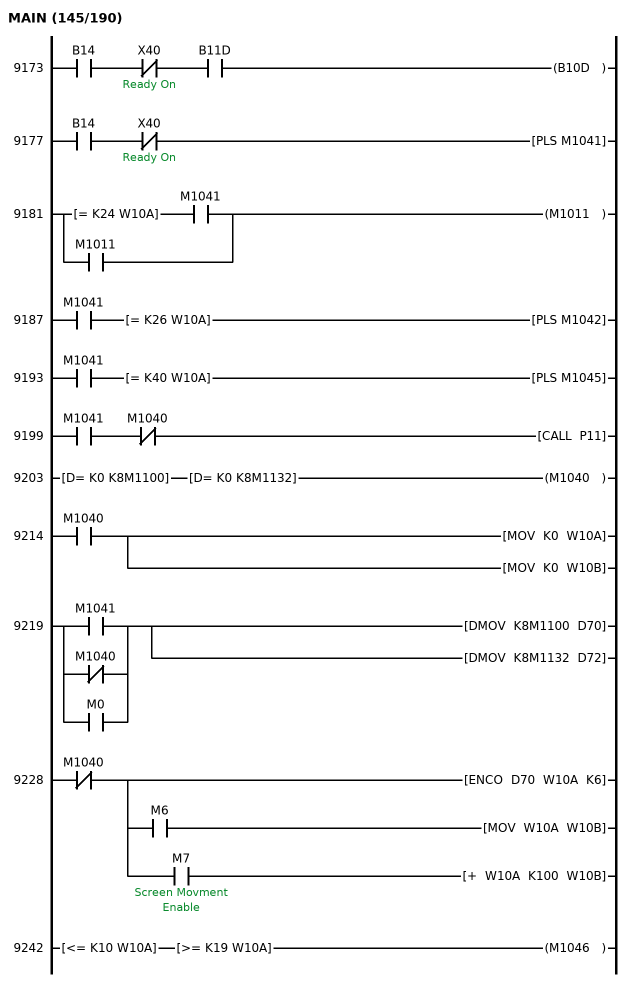
[picture p144: ladder of MAIN, rungs at steps 9173 to 9242]
9173  LD      B14
      ANI     X40  ; Ready On
      AND     B11D
      OUT     B10D
9177  LD      B14
      ANI     X40  ; Ready On
      PLS     M1041
9181  LD=     K24 W10A
      AND     M1041
      OR      M1011
      OUT     M1011
9187  LD      M1041
      AND=    K26 W10A
      PLS     M1042
9193  LD      M1041
      AND=    K40 W10A
      PLS     M1045
9199  LD      M1041
      ANI     M1040
      CALL    P11
9203  LDD=    K0 K8M1100
      ANDD=   K0 K8M1132
      OUT     M1040
9214  LD      M1040
      MOV     K0 W10A
      MOV     K0 W10B
9219  LD      M1041
      ORI     M1040
      OR      M0
      DMOV    K8M1100 D70
      DMOV    K8M1132 D72
9228  LDI     M1040
      ENCO    D70 W10A K6
      MPS
      AND     M6
      MOV     W10A W10B
      MPP
      AND     M7  ; Screen Movment Enable
      +       W10A K100 W10B
9242  LD<=    K10 W10A
      AND>=   K19 W10A
      OUT     M1046
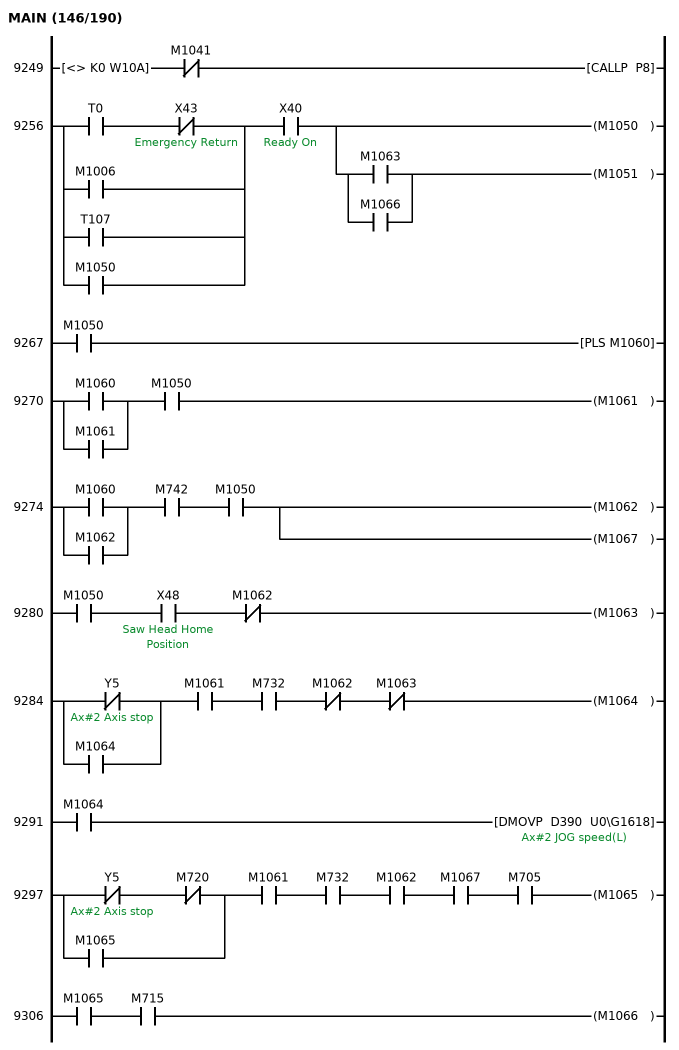
9249  LD<>    K0 W10A
      ANI     M1041
      CALLP   P8
9256  LD      T0
      ANI     X43  ; Emergency Return
      OR      M1006
      OR      T107
      OR      M1050
      AND     X40  ; Ready On
      OUT     M1050
      LD      M1063
      OR      M1066
      ANB
      OUT     M1051
9267  LD      M1050
      PLS     M1060
9270  LD      M1060
      OR      M1061
      AND     M1050
      OUT     M1061
9274  LD      M1060
      OR      M1062
      AND     M742
      AND     M1050
      OUT     M1062
      OUT     M1067
9280  LD      M1050
      AND     X48  ; Saw Head Home Position
      ANI     M1062
      OUT     M1063
9284  LDI     Y5  ; Ax#2 Axis stop
      OR      M1064
      AND     M1061
      AND     M732
      ANI     M1062
      ANI     M1063
      OUT     M1064
9291  LD      M1064
      DMOVP   D390 U0\G1618
9297  LDI     Y5  ; Ax#2 Axis stop
      ANI     M720
      OR      M1065
      AND     M1061
      AND     M732
      AND     M1062
      AND     M1067
      AND     M705
      OUT     M1065
9306  LD      M1065
      AND     M715
      OUT     M1066
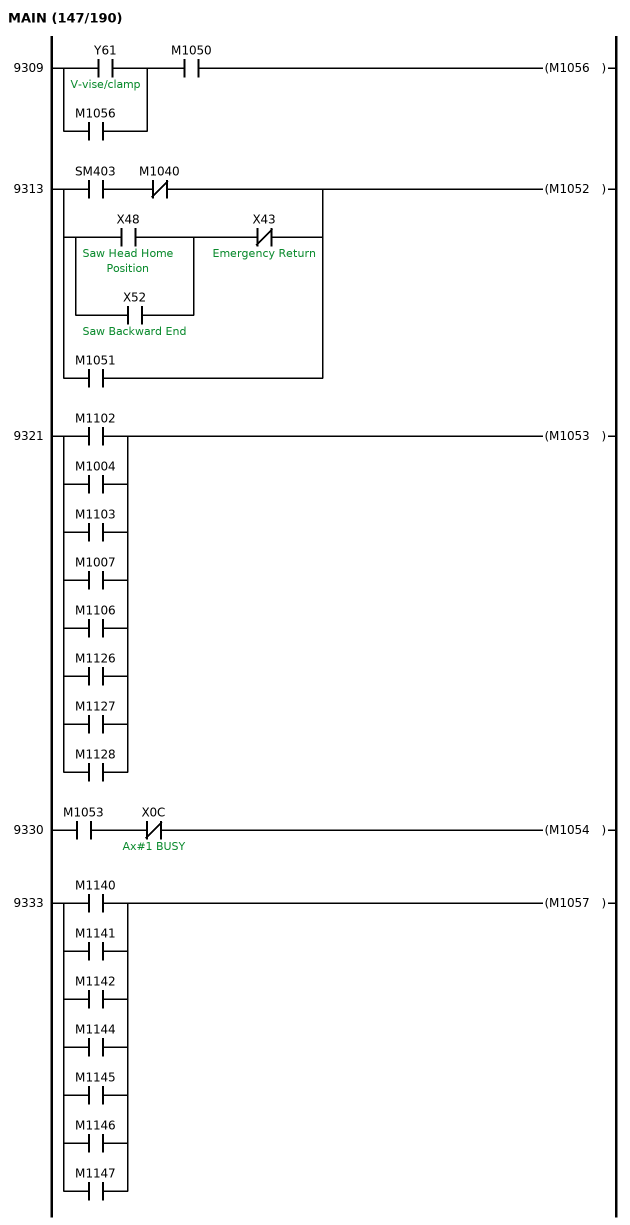
9309  LD      Y61  ; V-vise/clamp
      OR      M1056
      AND     M1050
      OUT     M1056
9313  LD      SM403
      ANI     M1040
      LD      X48  ; Saw Head Home Position
      OR      X52  ; Saw Backward End
      ANI     X43  ; Emergency Return
      ORB
      OR      M1051
      OUT     M1052
9321  LD      M1102
      OR      M1004
      OR      M1103
      OR      M1007
      OR      M1106
      OR      M1126
      OR      M1127
      OR      M1128
      OUT     M1053
9330  LD      M1053
      ANI     X0C  ; Ax#1 BUSY
      OUT     M1054
9333  LD      M1140
      OR      M1141
      OR      M1142
      OR      M1144
      OR      M1145
      OR      M1146
      OR      M1147
      OUT     M1057
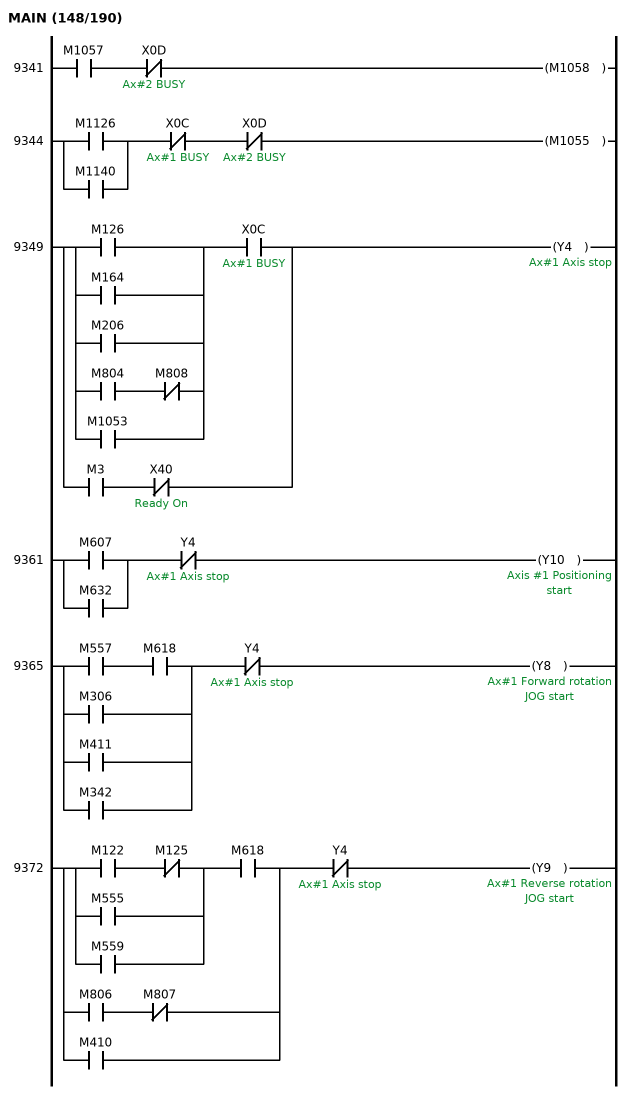
9341  LD      M1057
      ANI     X0D  ; Ax#2 BUSY
      OUT     M1058
9344  LD      M1126
      OR      M1140
      ANI     X0C  ; Ax#1 BUSY
      ANI     X0D  ; Ax#2 BUSY
      OUT     M1055
9349  LD      M126
      OR      M164
      OR      M206
      LD      M804
      ANI     M808
      ORB
      OR      M1053
      AND     X0C  ; Ax#1 BUSY
      LD      M3
      ANI     X40  ; Ready On
      ORB
      OUT     Y4  ; Ax#1 Axis stop
9361  LD      M607
      OR      M632
      ANI     Y4  ; Ax#1 Axis stop
      OUT     Y10  ; Axis #1 Positioning start
9365  LD      M557
      AND     M618
      OR      M306
      OR      M411
      OR      M342
      ANI     Y4  ; Ax#1 Axis stop
      OUT     Y8  ; Ax#1 Forward rotation JOG start
9372  LD      M122
      ANI     M125
      OR      M555
      OR      M559
      AND     M618
      LD      M806
      ANI     M807
      ORB
      OR      M410
      ANI     Y4  ; Ax#1 Axis stop
      OUT     Y9  ; Ax#1 Reverse rotation JOG start
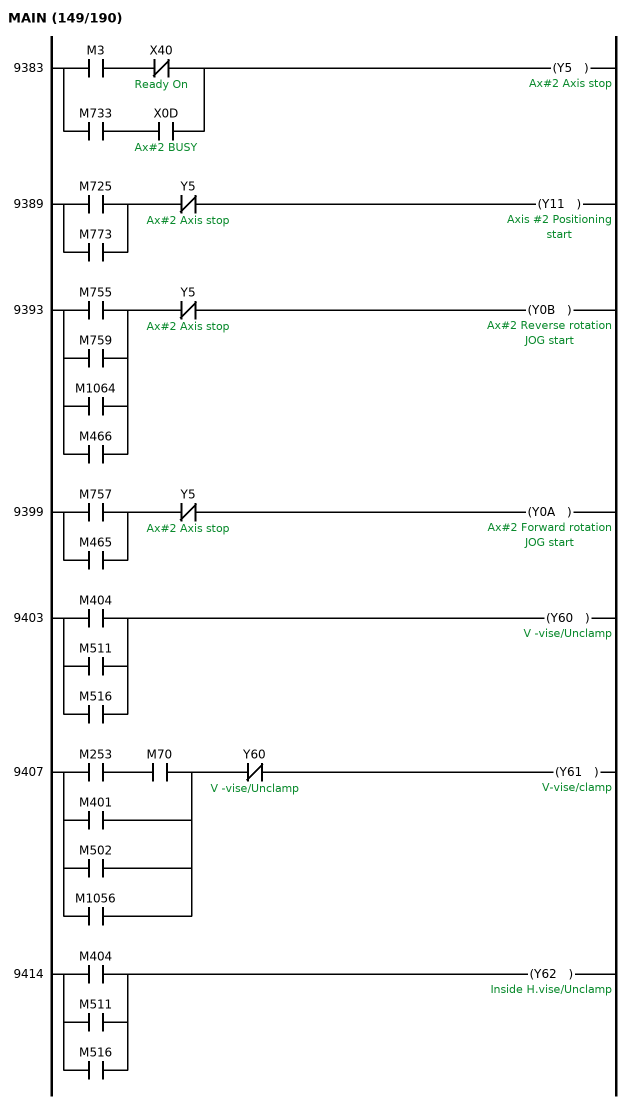
9383  LD      M3
      ANI     X40  ; Ready On
      LD      M733
      AND     X0D  ; Ax#2 BUSY
      ORB
      OUT     Y5  ; Ax#2 Axis stop
9389  LD      M725
      OR      M773
      ANI     Y5  ; Ax#2 Axis stop
      OUT     Y11  ; Axis #2 Positioning start
9393  LD      M755
      OR      M759
      OR      M1064
      OR      M466
      ANI     Y5  ; Ax#2 Axis stop
      OUT     Y0B  ; Ax#2 Reverse rotation JOG start
9399  LD      M757
      OR      M465
      ANI     Y5  ; Ax#2 Axis stop
      OUT     Y0A  ; Ax#2 Forward rotation JOG start
9403  LD      M404
      OR      M511
      OR      M516
      OUT     Y60  ; V -vise/Unclamp
9407  LD      M253
      AND     M70
      OR      M401
      OR      M502
      OR      M1056
      ANI     Y60  ; V -vise/Unclamp
      OUT     Y61  ; V-vise/clamp
9414  LD      M404
      OR      M511
      OR      M516
      OUT     Y62  ; Inside H.vise/Unclamp
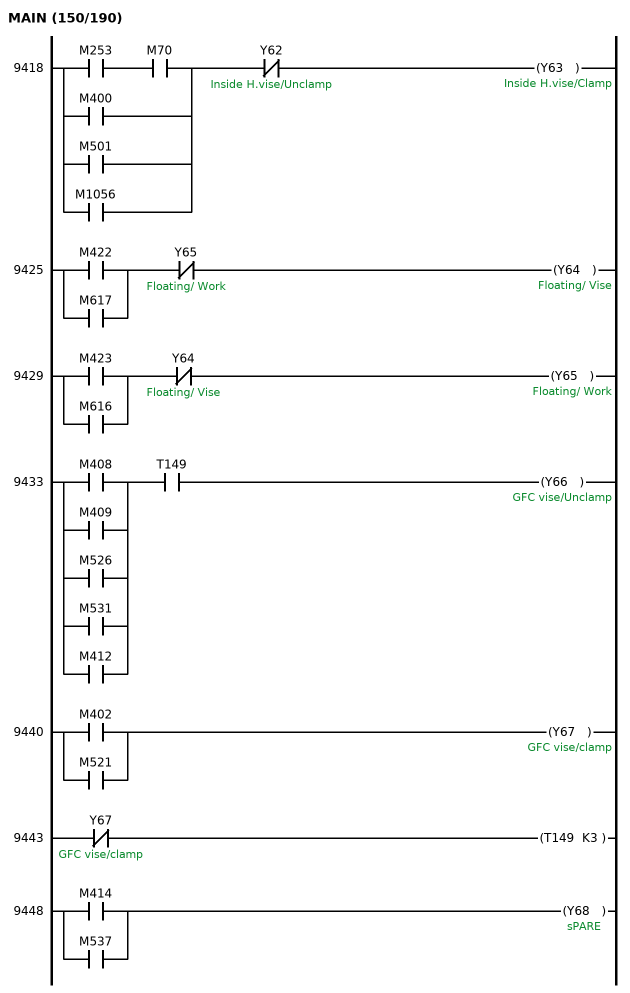
9418  LD      M253
      AND     M70
      OR      M400
      OR      M501
      OR      M1056
      ANI     Y62  ; Inside H.vise/Unclamp
      OUT     Y63  ; Inside H.vise/Clamp
9425  LD      M422
      OR      M617
      ANI     Y65  ; Floating/ Work
      OUT     Y64  ; Floating/ Vise
9429  LD      M423
      OR      M616
      ANI     Y64  ; Floating/ Vise
      OUT     Y65  ; Floating/ Work
9433  LD      M408
      OR      M409
      OR      M526
      OR      M531
      OR      M412
      AND     T149
      OUT     Y66  ; GFC vise/Unclamp
9440  LD      M402
      OR      M521
      OUT     Y67  ; GFC vise/clamp
9443  LDI     Y67  ; GFC vise/clamp
      OUT     T149 K3
9448  LD      M414
      OR      M537
      OUT     Y68  ; sPARE
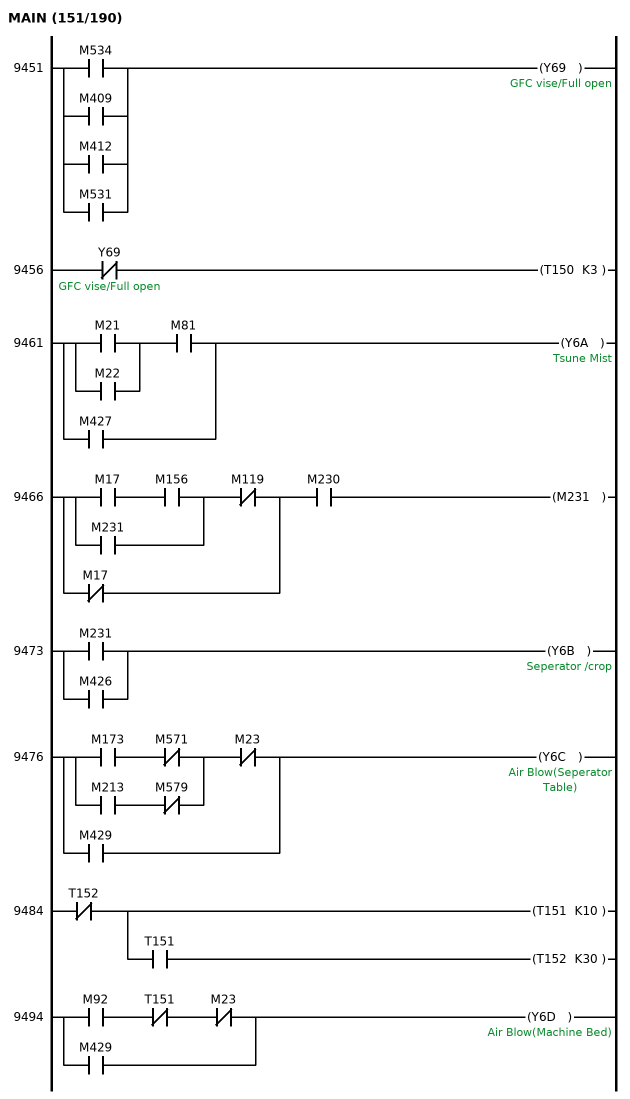
9451  LD      M534
      OR      M409
      OR      M412
      OR      M531
      OUT     Y69  ; GFC vise/Full open
9456  LDI     Y69  ; GFC vise/Full open
      OUT     T150 K3
9461  LD      M21
      OR      M22
      AND     M81
      OR      M427
      OUT     Y6A  ; Tsune Mist
9466  LD      M17
      AND     M156
      OR      M231
      ANI     M119
      ORI     M17
      AND     M230
      OUT     M231
9473  LD      M231
      OR      M426
      OUT     Y6B  ; Seperator /crop
9476  LD      M173
      ANI     M571
      LD      M213
      ANI     M579
      ORB
      ANI     M23
      OR      M429
      OUT     Y6C  ; Air Blow(Seperator Table)
9484  LDI     T152
      OUT     T151 K10
      AND     T151
      OUT     T152 K30
9494  LD      M92
      ANI     T151
      ANI     M23
      OR      M429
      OUT     Y6D  ; Air Blow(Machine Bed)
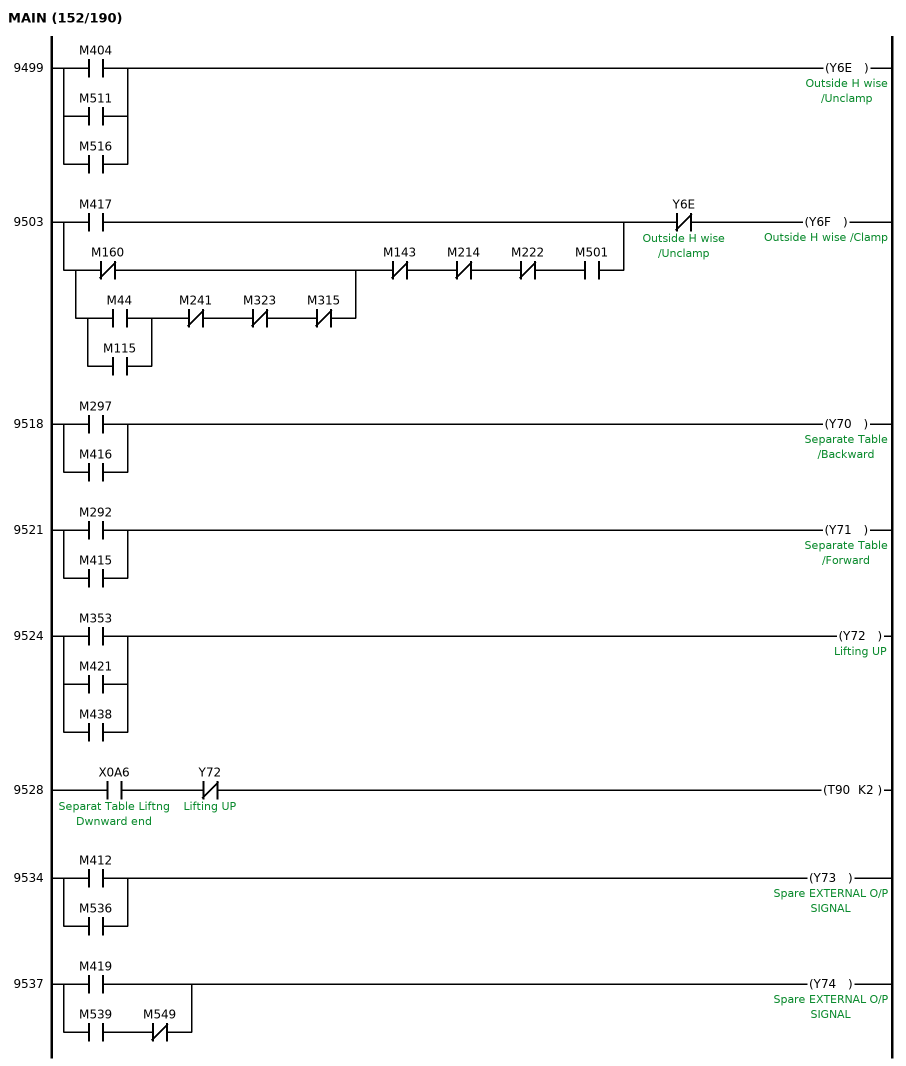
9499  LD      M404
      OR      M511
      OR      M516
      OUT     Y6E  ; Outside H wise /Unclamp
9503  LD      M417
      LDI     M160
      LD      M44
      OR      M115
      ANI     M241
      ANI     M323
      ANI     M315
      ORB
      ANI     M143
      ANI     M214
      ANI     M222
      AND     M501
      ORB
      ANI     Y6E  ; Outside H wise /Unclamp
      OUT     Y6F  ; Outside H wise /Clamp
9518  LD      M297
      OR      M416
      OUT     Y70  ; Separate Table /Backward
9521  LD      M292
      OR      M415
      OUT     Y71  ; Separate Table /Forward
9524  LD      M353
      OR      M421
      OR      M438
      OUT     Y72  ; Lifting UP
9528  LD      X0A6  ; Separat Table Liftng Dwnward end
      ANI     Y72  ; Lifting UP
      OUT     T90 K2
9534  LD      M412
      OR      M536
      OUT     Y73  ; Spare EXTERNAL O/P SIGNAL
9537  LD      M419
      LD      M539
      ANI     M549
      ORB
      OUT     Y74  ; Spare EXTERNAL O/P SIGNAL
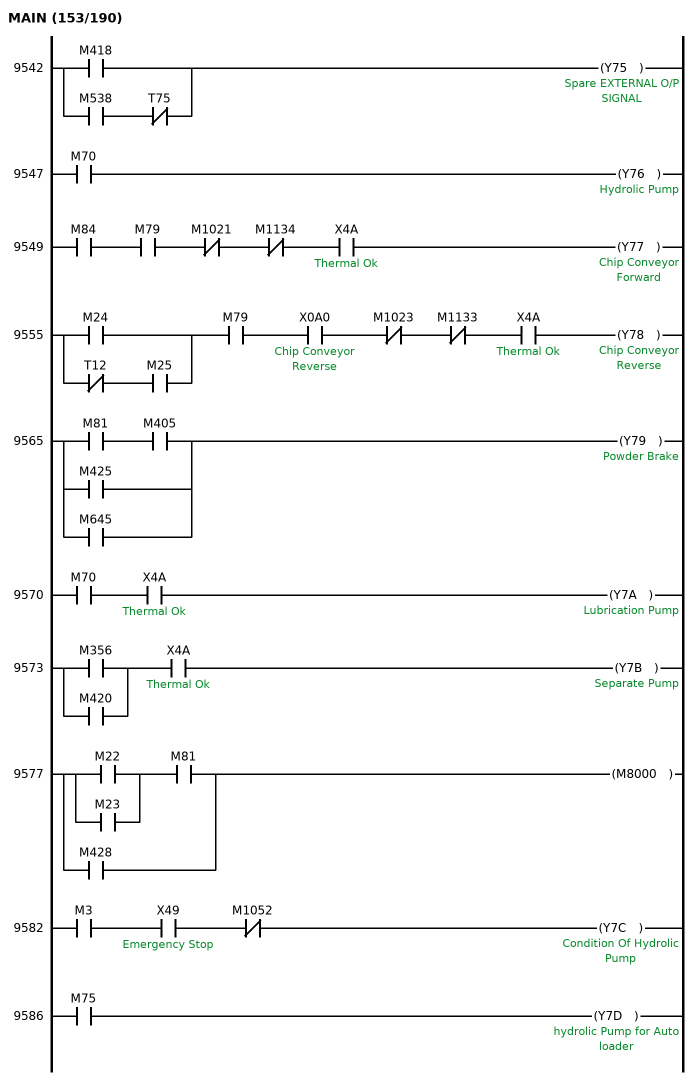
9542  LD      M418
      LD      M538
      ANI     T75
      ORB
      OUT     Y75  ; Spare EXTERNAL O/P SIGNAL
9547  LD      M70
      OUT     Y76  ; Hydrolic Pump
9549  LD      M84
      AND     M79
      ANI     M1021
      ANI     M1134
      AND     X4A  ; Thermal Ok
      OUT     Y77  ; Chip Conveyor Forward
9555  LD      M24
      LDI     T12
      AND     M25
      ORB
      AND     M79
      AND     X0A0  ; Chip Conveyor Reverse
      ANI     M1023
      ANI     M1133
      AND     X4A  ; Thermal Ok
      OUT     Y78  ; Chip Conveyor Reverse
9565  LD      M81
      AND     M405
      OR      M425
      OR      M645
      OUT     Y79  ; Powder Brake
9570  LD      M70
      AND     X4A  ; Thermal Ok
      OUT     Y7A  ; Lubrication Pump
9573  LD      M356
      OR      M420
      AND     X4A  ; Thermal Ok
      OUT     Y7B  ; Separate Pump
9577  LD      M22
      OR      M23
      AND     M81
      OR      M428
      OUT     M8000
9582  LD      M3
      AND     X49  ; Emergency Stop
      ANI     M1052
      OUT     Y7C  ; Condition Of Hydrolic Pump
9586  LD      M75
      OUT     Y7D  ; hydrolic Pump for Auto loader
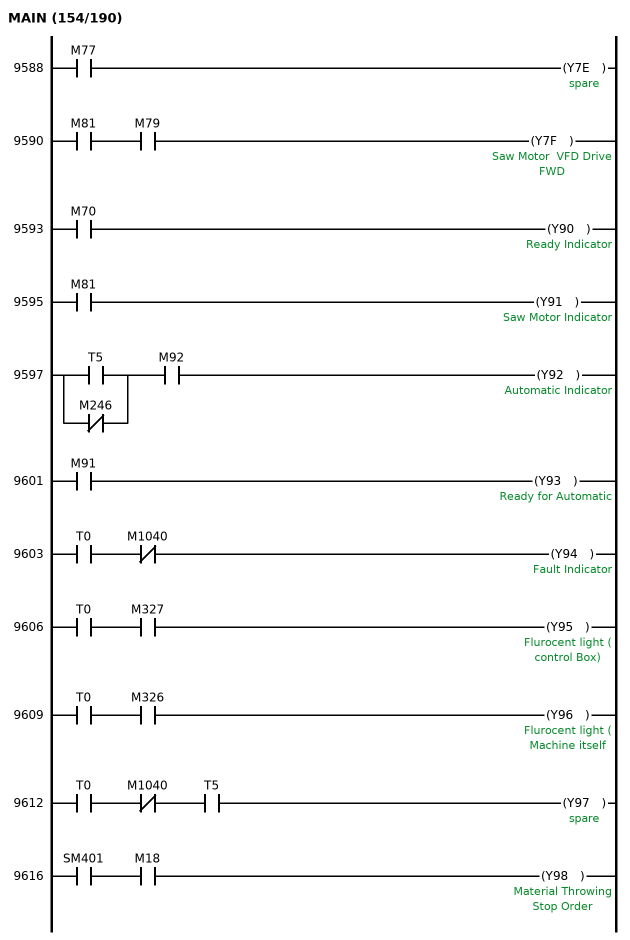
9588  LD      M77
      OUT     Y7E  ; spare
9590  LD      M81
      AND     M79
      OUT     Y7F  ; Saw Motor  VFD Drive FWD
9593  LD      M70
      OUT     Y90  ; Ready Indicator
9595  LD      M81
      OUT     Y91  ; Saw Motor Indicator
9597  LD      T5
      ORI     M246
      AND     M92
      OUT     Y92  ; Automatic Indicator
9601  LD      M91
      OUT     Y93  ; Ready for Automatic
9603  LD      T0
      ANI     M1040
      OUT     Y94  ; Fault Indicator
9606  LD      T0
      AND     M327
      OUT     Y95  ; Flurocent light ( control Box)
9609  LD      T0
      AND     M326
      OUT     Y96  ; Flurocent light ( Machine itself
9612  LD      T0
      ANI     M1040
      AND     T5
      OUT     Y97  ; spare
9616  LD      SM401
      AND     M18
      OUT     Y98  ; Material Throwing Stop Order
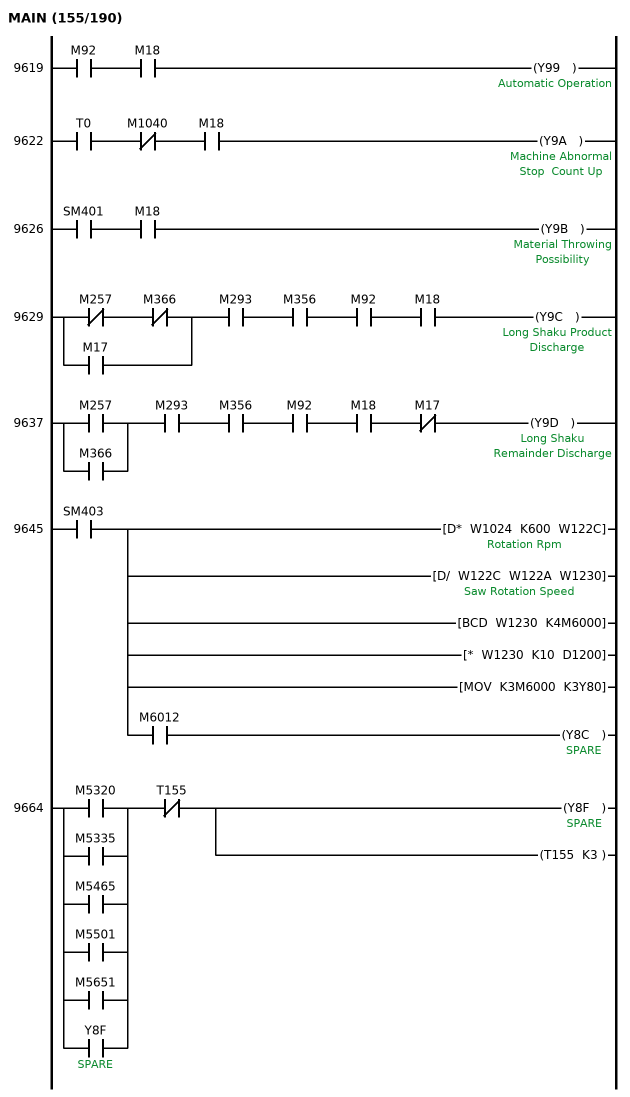
9619  LD      M92
      AND     M18
      OUT     Y99  ; Automatic Operation
9622  LD      T0
      ANI     M1040
      AND     M18
      OUT     Y9A  ; Machine Abnormal Stop  Count Up
9626  LD      SM401
      AND     M18
      OUT     Y9B  ; Material Throwing Possibility
9629  LDI     M257
      ANI     M366
      OR      M17
      AND     M293
      AND     M356
      AND     M92
      AND     M18
      OUT     Y9C  ; Long Shaku Product Discharge
9637  LD      M257
      OR      M366
      AND     M293
      AND     M356
      AND     M92
      AND     M18
      ANI     M17
      OUT     Y9D  ; Long Shaku Remainder Discharge
9645  LD      SM403
      D*      W1024 K600 W122C
      D/      W122C W122A W1230  ; Saw Rotation Speed
      BCD     W1230 K4M6000
      *       W1230 K10 D1200
      MOV     K3M6000 K3Y80  ; SPARE
      AND     M6012
      OUT     Y8C  ; SPARE
9664  LD      M5320
      OR      M5335
      OR      M5465
      OR      M5501
      OR      M5651
      OR      Y8F  ; SPARE
      ANI     T155
      OUT     Y8F  ; SPARE
      OUT     T155 K3
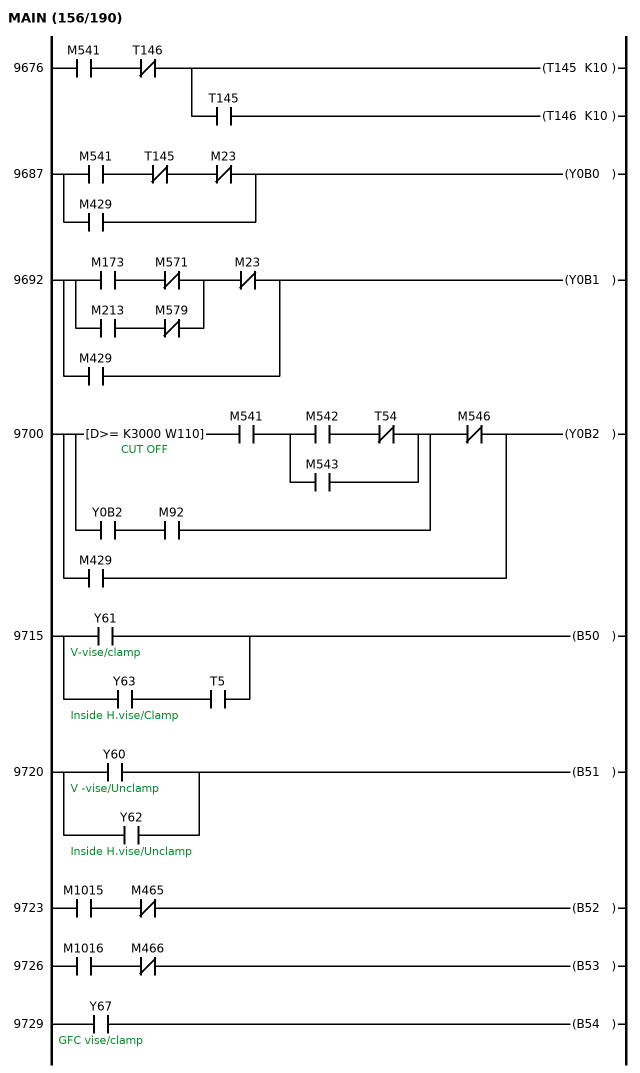
9676  LD      M541
      ANI     T146
      OUT     T145 K10
      AND     T145
      OUT     T146 K10
9687  LD      M541
      ANI     T145
      ANI     M23
      OR      M429
      OUT     Y0B0
9692  LD      M173
      ANI     M571
      LD      M213
      ANI     M579
      ORB
      ANI     M23
      OR      M429
      OUT     Y0B1
9700  LDD>=   K3000 W110  ; CUT OFF
      AND     M541
      LD      M542
      ANI     T54
      OR      M543
      ANB
      LD      Y0B2
      AND     M92
      ORB
      ANI     M546
      OR      M429
      OUT     Y0B2
9715  LD      Y61  ; V-vise/clamp
      LD      Y63  ; Inside H.vise/Clamp
      AND     T5
      ORB
      OUT     B50
9720  LD      Y60  ; V -vise/Unclamp
      OR      Y62  ; Inside H.vise/Unclamp
      OUT     B51
9723  LD      M1015
      ANI     M465
      OUT     B52
9726  LD      M1016
      ANI     M466
      OUT     B53
9729  LD      Y67  ; GFC vise/clamp
      OUT     B54
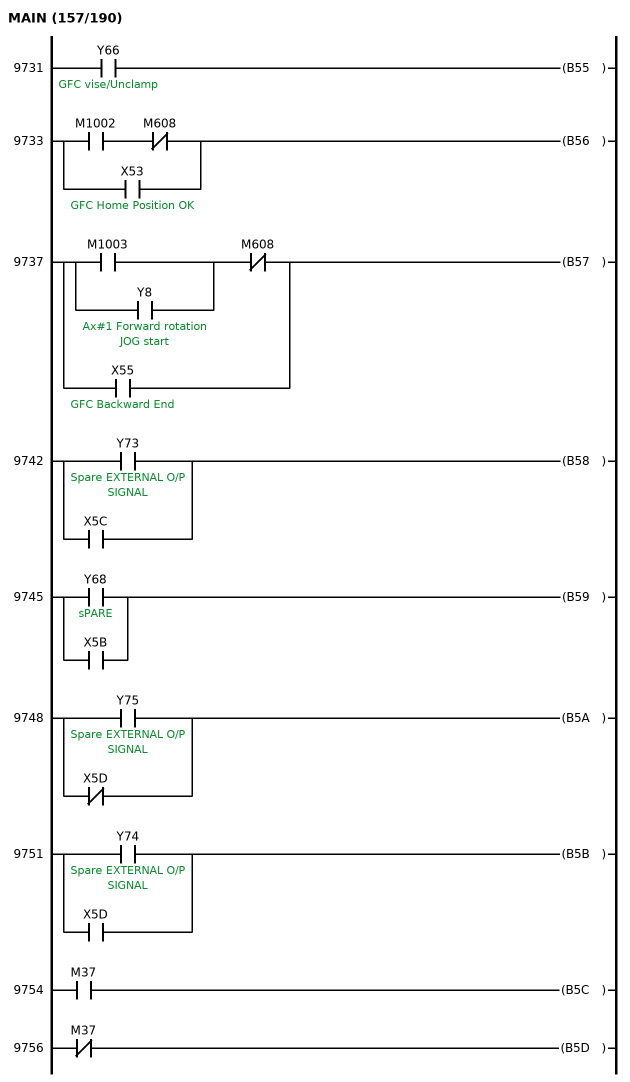
9731  LD      Y66  ; GFC vise/Unclamp
      OUT     B55
9733  LD      M1002
      ANI     M608
      OR      X53  ; GFC Home Position OK
      OUT     B56
9737  LD      M1003
      OR      Y8  ; Ax#1 Forward rotation JOG start
      ANI     M608
      OR      X55  ; GFC Backward End
      OUT     B57
9742  LD      Y73  ; Spare EXTERNAL O/P SIGNAL
      OR      X5C
      OUT     B58
9745  LD      Y68  ; sPARE
      OR      X5B
      OUT     B59
9748  LD      Y75  ; Spare EXTERNAL O/P SIGNAL
      ORI     X5D
      OUT     B5A
9751  LD      Y74  ; Spare EXTERNAL O/P SIGNAL
      OR      X5D
      OUT     B5B
9754  LD      M37
      OUT     B5C
9756  LDI     M37
      OUT     B5D
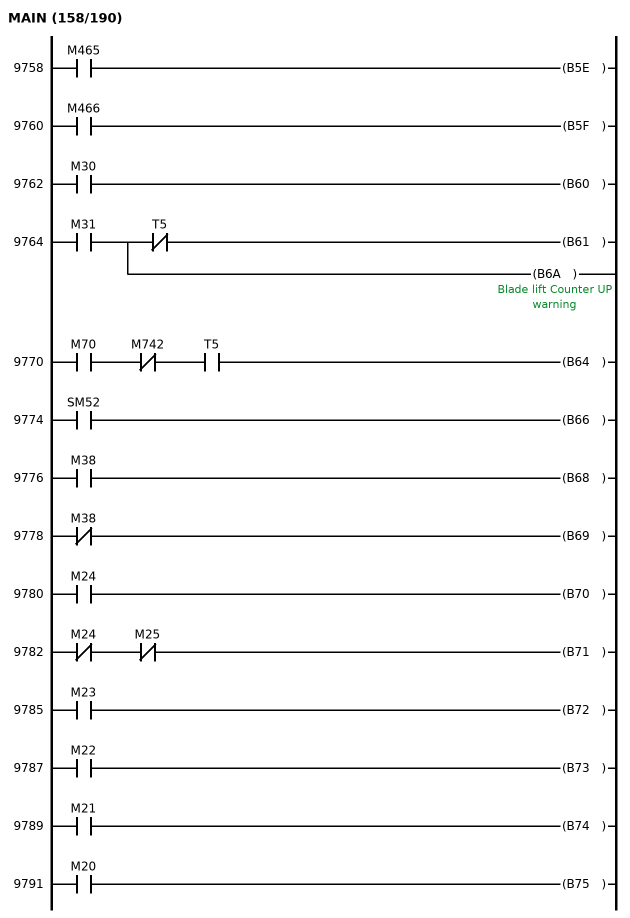
9758  LD      M465
      OUT     B5E
9760  LD      M466
      OUT     B5F
9762  LD      M30
      OUT     B60
9764  LD      M31
      MPS
      ANI     T5
      OUT     B61
      MPP
      OUT     B6A  ; Blade lift Counter UP warning
9770  LD      M70
      ANI     M742
      AND     T5
      OUT     B64
9774  LD      SM52
      OUT     B66
9776  LD      M38
      OUT     B68
9778  LDI     M38
      OUT     B69
9780  LD      M24
      OUT     B70
9782  LDI     M24
      ANI     M25
      OUT     B71
9785  LD      M23
      OUT     B72
9787  LD      M22
      OUT     B73
9789  LD      M21
      OUT     B74
9791  LD      M20
      OUT     B75
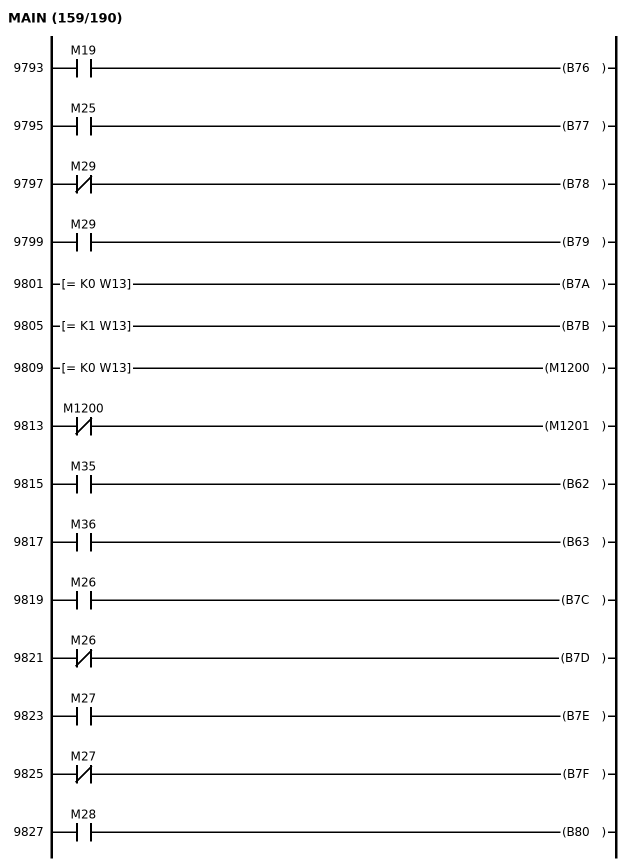
9793  LD      M19
      OUT     B76
9795  LD      M25
      OUT     B77
9797  LDI     M29
      OUT     B78
9799  LD      M29
      OUT     B79
9801  LD=     K0 W13
      OUT     B7A
9805  LD=     K1 W13
      OUT     B7B
9809  LD=     K0 W13
      OUT     M1200
9813  LDI     M1200
      OUT     M1201
9815  LD      M35
      OUT     B62
9817  LD      M36
      OUT     B63
9819  LD      M26
      OUT     B7C
9821  LDI     M26
      OUT     B7D
9823  LD      M27
      OUT     B7E
9825  LDI     M27
      OUT     B7F
9827  LD      M28
      OUT     B80
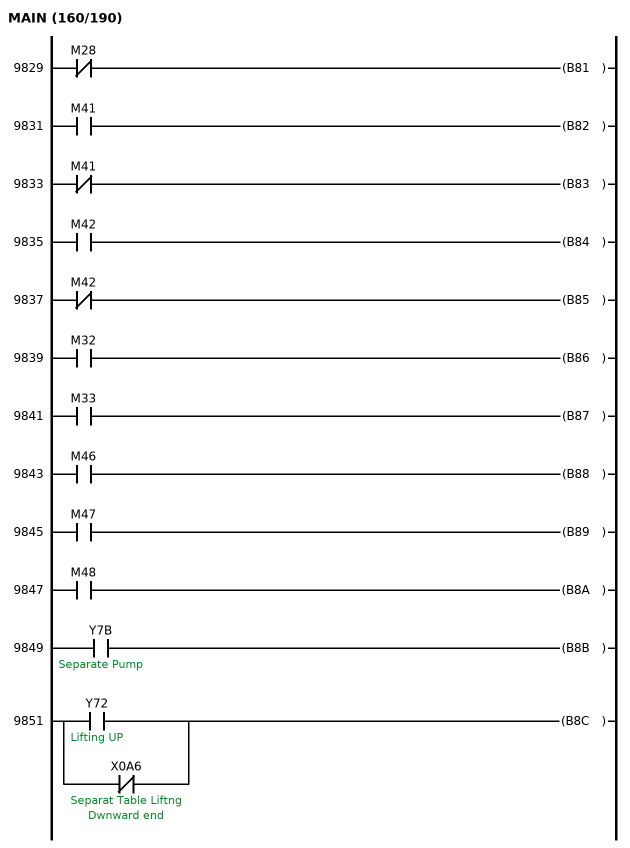
9829  LDI     M28
      OUT     B81
9831  LD      M41
      OUT     B82
9833  LDI     M41
      OUT     B83
9835  LD      M42
      OUT     B84
9837  LDI     M42
      OUT     B85
9839  LD      M32
      OUT     B86
9841  LD      M33
      OUT     B87
9843  LD      M46
      OUT     B88
9845  LD      M47
      OUT     B89
9847  LD      M48
      OUT     B8A
9849  LD      Y7B  ; Separate Pump
      OUT     B8B
9851  LD      Y72  ; Lifting UP
      ORI     X0A6  ; Separat Table Liftng Dwnward end
      OUT     B8C
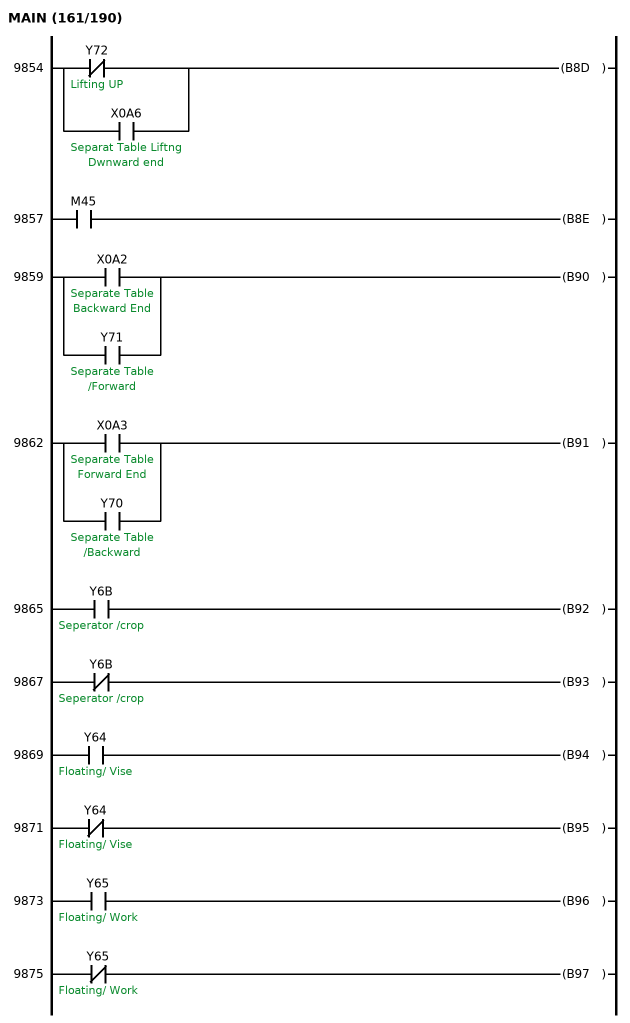
9854  LDI     Y72  ; Lifting UP
      OR      X0A6  ; Separat Table Liftng Dwnward end
      OUT     B8D
9857  LD      M45
      OUT     B8E
9859  LD      X0A2  ; Separate Table Backward End
      OR      Y71  ; Separate Table /Forward
      OUT     B90
9862  LD      X0A3  ; Separate Table Forward End
      OR      Y70  ; Separate Table /Backward
      OUT     B91
9865  LD      Y6B  ; Seperator /crop
      OUT     B92
9867  LDI     Y6B  ; Seperator /crop
      OUT     B93
9869  LD      Y64  ; Floating/ Vise
      OUT     B94
9871  LDI     Y64  ; Floating/ Vise
      OUT     B95
9873  LD      Y65  ; Floating/ Work
      OUT     B96
9875  LDI     Y65  ; Floating/ Work
      OUT     B97
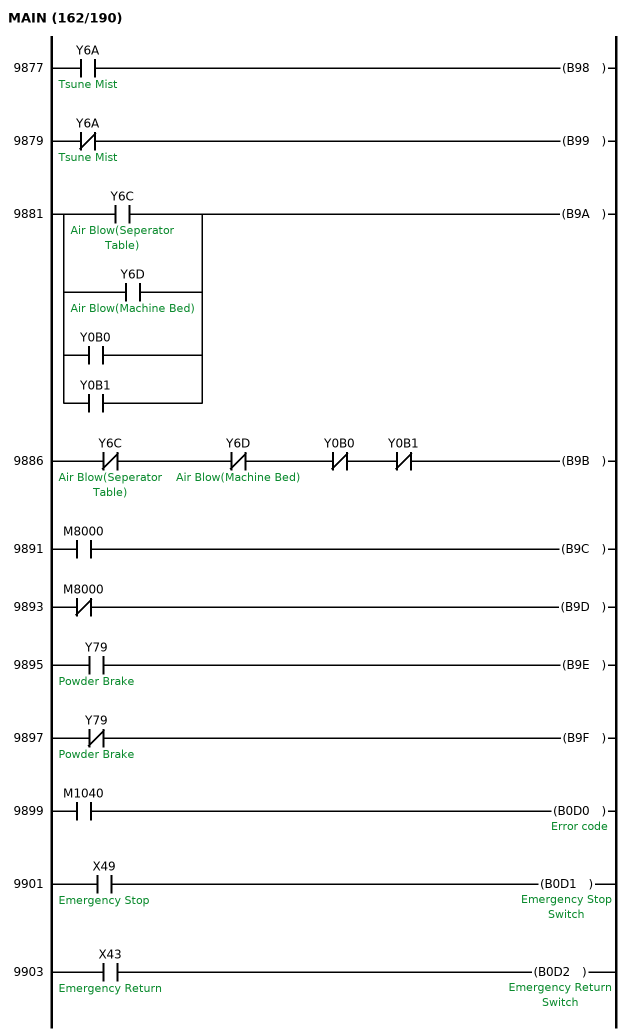
9877  LD      Y6A  ; Tsune Mist
      OUT     B98
9879  LDI     Y6A  ; Tsune Mist
      OUT     B99
9881  LD      Y6C  ; Air Blow(Seperator Table)
      OR      Y6D  ; Air Blow(Machine Bed)
      OR      Y0B0
      OR      Y0B1
      OUT     B9A
9886  LDI     Y6C  ; Air Blow(Seperator Table)
      ANI     Y6D  ; Air Blow(Machine Bed)
      ANI     Y0B0
      ANI     Y0B1
      OUT     B9B
9891  LD      M8000
      OUT     B9C
9893  LDI     M8000
      OUT     B9D
9895  LD      Y79  ; Powder Brake
      OUT     B9E
9897  LDI     Y79  ; Powder Brake
      OUT     B9F
9899  LD      M1040
      OUT     B0D0  ; Error code
9901  LD      X49  ; Emergency Stop
      OUT     B0D1  ; Emergency Stop Switch
9903  LD      X43  ; Emergency Return
      OUT     B0D2  ; Emergency Return Switch
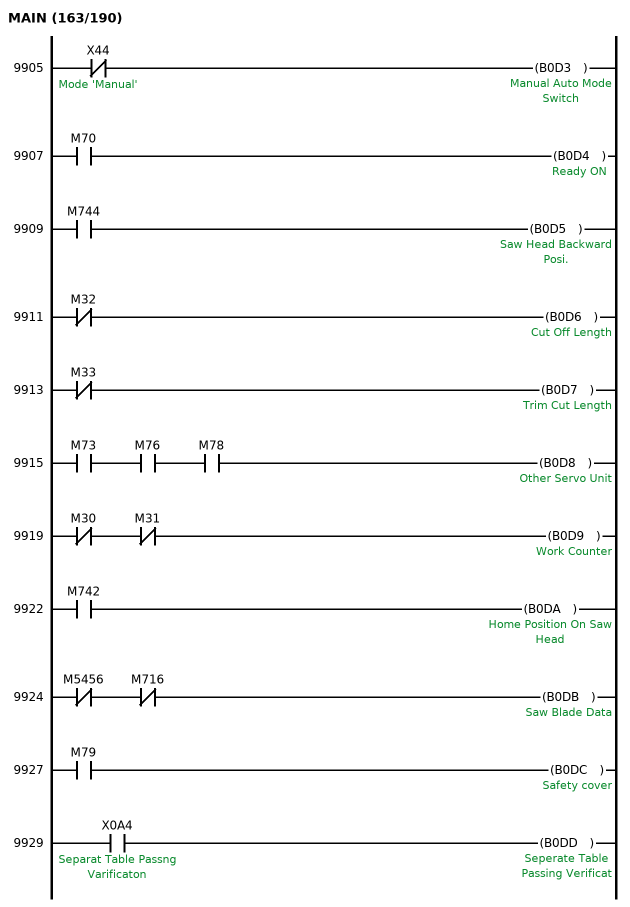
9905  LDI     X44  ; Mode 'Manual'
      OUT     B0D3  ; Manual Auto Mode Switch
9907  LD      M70
      OUT     B0D4  ; Ready ON
9909  LD      M744
      OUT     B0D5  ; Saw Head Backward Posi.
9911  LDI     M32
      OUT     B0D6  ; Cut Off Length
9913  LDI     M33
      OUT     B0D7  ; Trim Cut Length
9915  LD      M73
      AND     M76
      AND     M78
      OUT     B0D8  ; Other Servo Unit
9919  LDI     M30
      ANI     M31
      OUT     B0D9  ; Work Counter
9922  LD      M742
      OUT     B0DA  ; Home Position On Saw Head
9924  LDI     M5456
      ANI     M716
      OUT     B0DB  ; Saw Blade Data
9927  LD      M79
      OUT     B0DC  ; Safety cover
9929  LD      X0A4  ; Separat Table Passng Varificaton
      OUT     B0DD  ; Seperate Table Passing Verificat
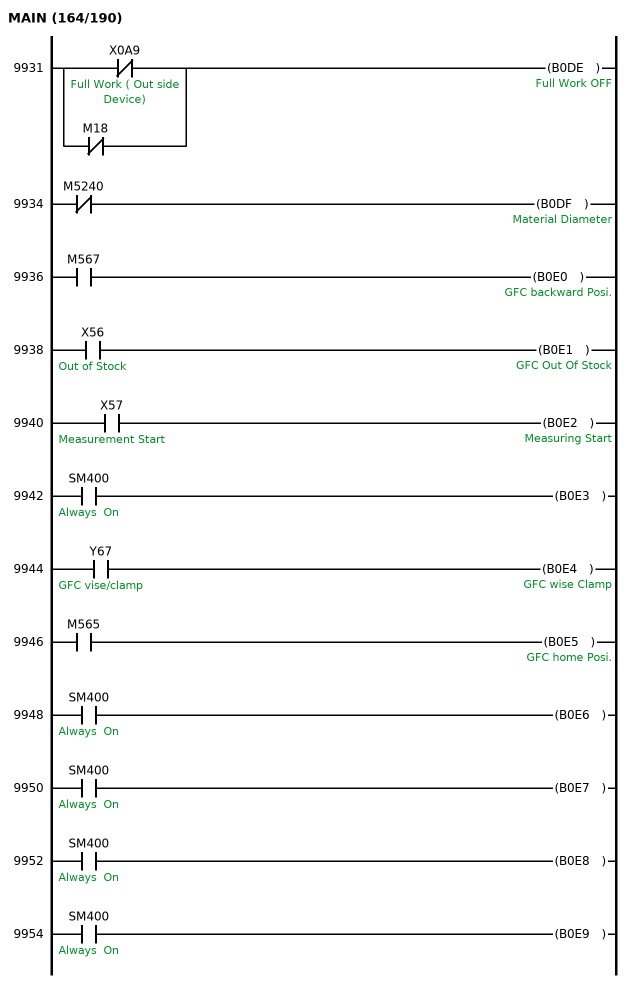
9931  LDI     X0A9  ; Full Work ( Out side Device)
      ORI     M18
      OUT     B0DE  ; Full Work OFF
9934  LDI     M5240
      OUT     B0DF  ; Material Diameter
9936  LD      M567
      OUT     B0E0  ; GFC backward Posi.
9938  LD      X56  ; Out of Stock
      OUT     B0E1  ; GFC Out Of Stock
9940  LD      X57  ; Measurement Start
      OUT     B0E2  ; Measuring Start
9942  LD      SM400  ; Always  On
      OUT     B0E3
9944  LD      Y67  ; GFC vise/clamp
      OUT     B0E4  ; GFC wise Clamp
9946  LD      M565
      OUT     B0E5  ; GFC home Posi.
9948  LD      SM400  ; Always  On
      OUT     B0E6
9950  LD      SM400  ; Always  On
      OUT     B0E7
9952  LD      SM400  ; Always  On
      OUT     B0E8
9954  LD      SM400  ; Always  On
      OUT     B0E9
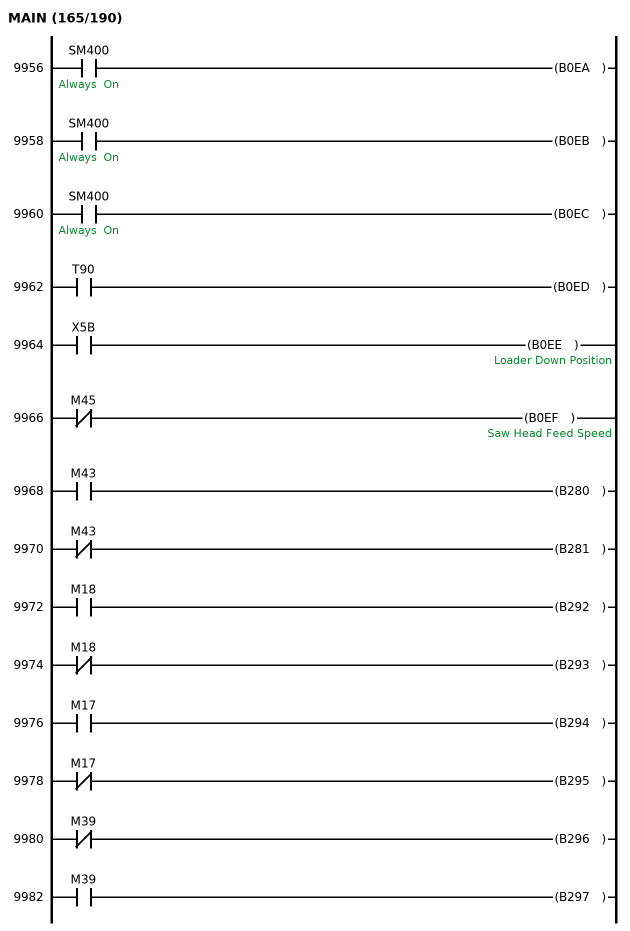
9956  LD      SM400  ; Always  On
      OUT     B0EA
9958  LD      SM400  ; Always  On
      OUT     B0EB
9960  LD      SM400  ; Always  On
      OUT     B0EC
9962  LD      T90
      OUT     B0ED
9964  LD      X5B
      OUT     B0EE  ; Loader Down Position
9966  LDI     M45
      OUT     B0EF  ; Saw Head Feed Speed
9968  LD      M43
      OUT     B280
9970  LDI     M43
      OUT     B281
9972  LD      M18
      OUT     B292
9974  LDI     M18
      OUT     B293
9976  LD      M17
      OUT     B294
9978  LDI     M17
      OUT     B295
9980  LDI     M39
      OUT     B296
9982  LD      M39
      OUT     B297
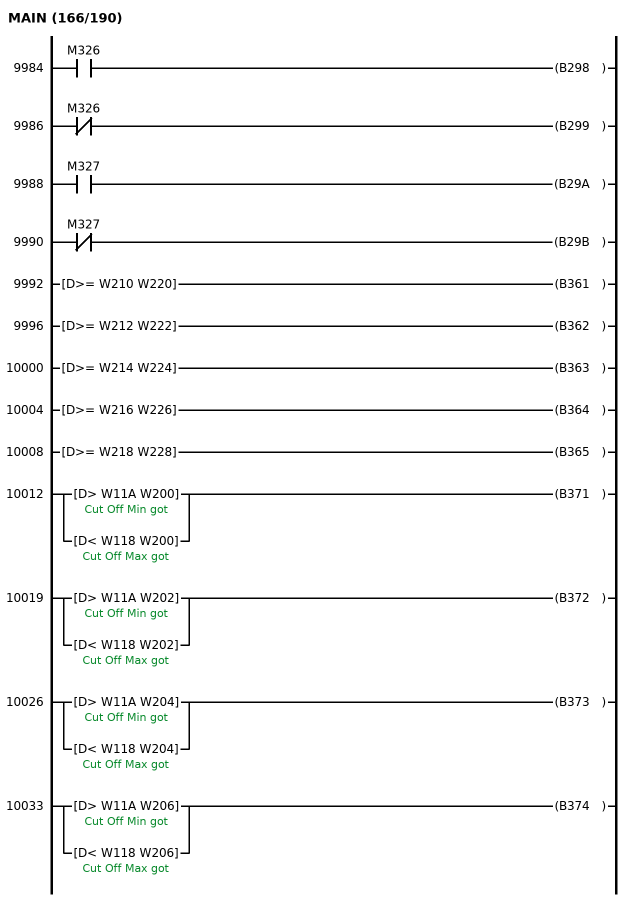
9984  LD      M326
      OUT     B298
9986  LDI     M326
      OUT     B299
9988  LD      M327
      OUT     B29A
9990  LDI     M327
      OUT     B29B
9992  LDD>=   W210 W220
      OUT     B361
9996  LDD>=   W212 W222
      OUT     B362
10000 LDD>=   W214 W224
      OUT     B363
10004 LDD>=   W216 W226
      OUT     B364
10008 LDD>=   W218 W228
      OUT     B365
10012 LDD>    W11A W200  ; Cut Off Min got
      ORD<    W118 W200  ; Cut Off Max got
      OUT     B371
10019 LDD>    W11A W202  ; Cut Off Min got
      ORD<    W118 W202  ; Cut Off Max got
      OUT     B372
10026 LDD>    W11A W204  ; Cut Off Min got
      ORD<    W118 W204  ; Cut Off Max got
      OUT     B373
10033 LDD>    W11A W206  ; Cut Off Min got
      ORD<    W118 W206  ; Cut Off Max got
      OUT     B374
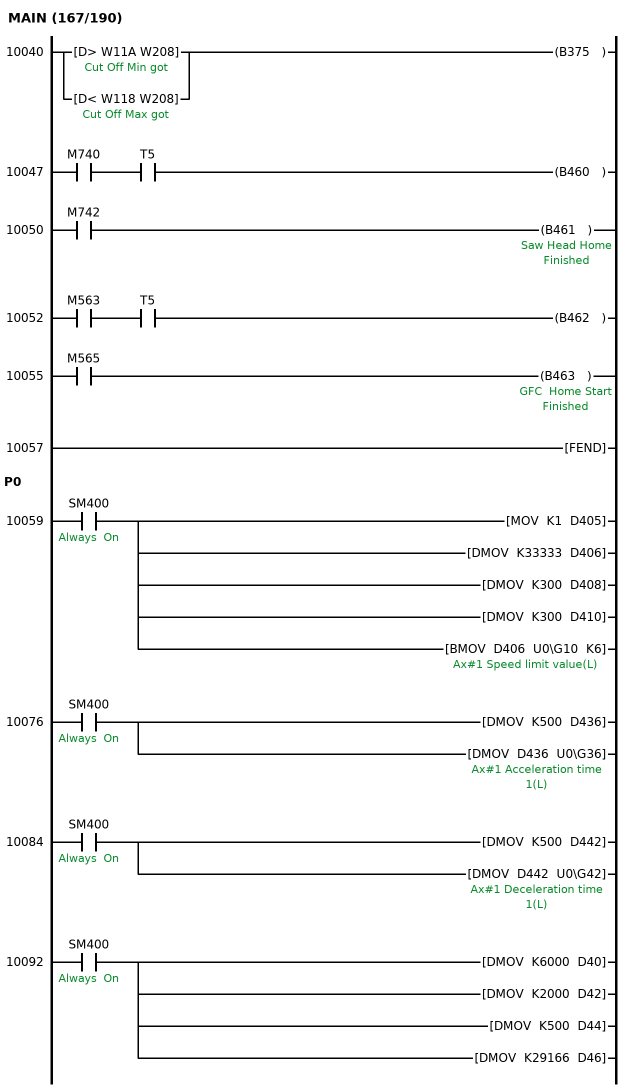
10040 LDD>    W11A W208  ; Cut Off Min got
      ORD<    W118 W208  ; Cut Off Max got
      OUT     B375
10047 LD      M740
      AND     T5
      OUT     B460
10050 LD      M742
      OUT     B461  ; Saw Head Home Finished
10052 LD      M563
      AND     T5
      OUT     B462
10055 LD      M565
      OUT     B463  ; GFC  Home Start Finished
10057 FEND
      P0
10059 LD      SM400  ; Always  On
      MOV     K1 D405
      DMOV    K33333 D406
      DMOV    K300 D408
      DMOV    K300 D410
      BMOV    D406 U0\G10 K6  ; Ax#1 Speed limit value(L)
10076 LD      SM400  ; Always  On
      DMOV    K500 D436
      DMOV    D436 U0\G36  ; Ax#1 Acceleration time 1(L)
10084 LD      SM400  ; Always  On
      DMOV    K500 D442
      DMOV    D442 U0\G42  ; Ax#1 Deceleration time 1(L)
10092 LD      SM400  ; Always  On
      DMOV    K6000 D40
      DMOV    K2000 D42
      DMOV    K500 D44
      DMOV    K29166 D46
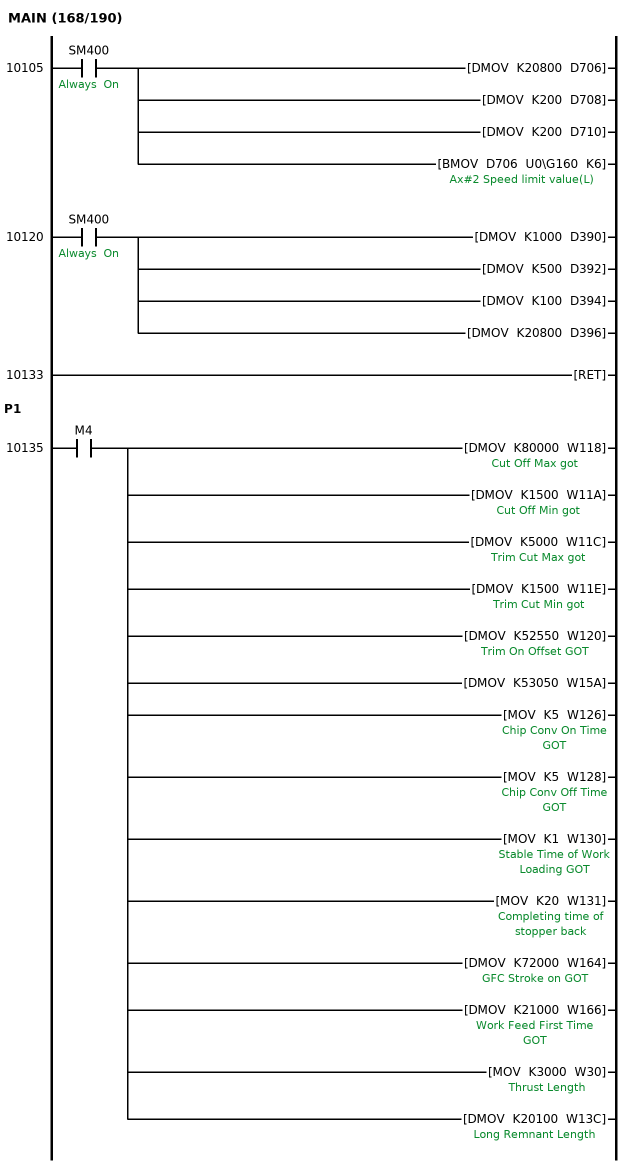
10105 LD      SM400  ; Always  On
      DMOV    K20800 D706
      DMOV    K200 D708
      DMOV    K200 D710
      BMOV    D706 U0\G160 K6  ; Ax#2 Speed limit value(L)
10120 LD      SM400  ; Always  On
      DMOV    K1000 D390
      DMOV    K500 D392
      DMOV    K100 D394
      DMOV    K20800 D396
10133 RET
      P1
10135 LD      M4
      DMOV    K80000 W118
      DMOV    K1500 W11A
      DMOV    K5000 W11C
      DMOV    K1500 W11E
      DMOV    K52550 W120
      DMOV    K53050 W15A
      MOV     K5 W126
      MOV     K5 W128
      MOV     K1 W130
      MOV     K20 W131
      DMOV    K72000 W164  ; GFC Stroke on GOT
      DMOV    K21000 W166  ; Work Feed First Time GOT
      MOV     K3000 W30
      DMOV    K20100 W13C
